% RSLogix 500 project Intro to PLC Job HO4 Greg.RSS, saved by version 10.00.00.00 %
PROJECT "UNTITLED"    % processor: Bul.1763 MicroLogix 1100 Series B %

PROGRAM FILES
  LAD 2   9 rungs

DATA FILES
  O0 OUTPUT  4 elements
  I1 INPUT  6 elements
  S2 STATUS  66 elements
  B3 BINARY  1 elements
  T4 TIMER  1 elements
  C5 COUNTER  1 elements
  R6 CONTROL  1 elements
  N7 INTEGER  1 elements
  F8 FLOAT  1 elements

LADDER 2
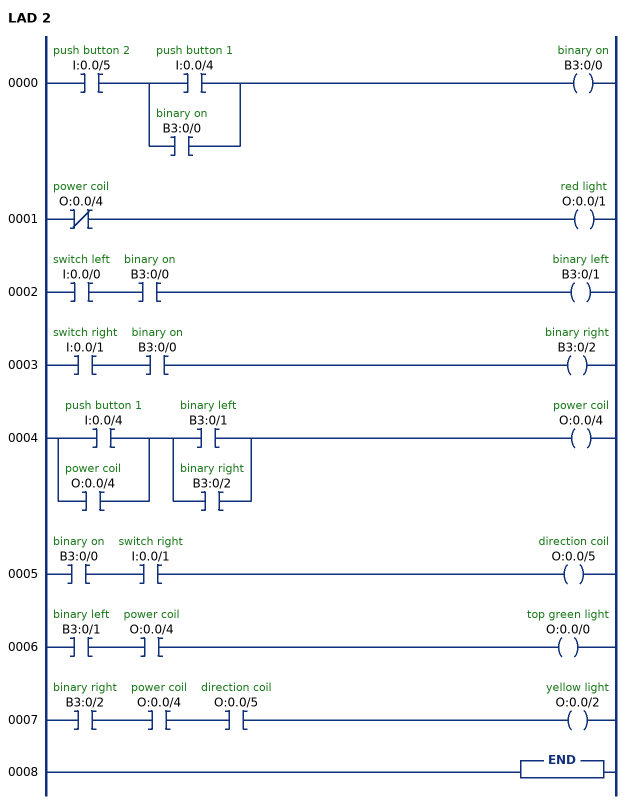
% Rung: 0 %
SOR XIC I:0.0/5 BST XIC I:0.0/4 NXB XIC B3:0/0 BND OTE B3:0/0 EOR
%   I:0.0/5  "push button 2" %
%   I:0.0/4  "push button 1" %
%   B3:0/0  "binary on" %
% Rung: 1 %
SOR XIO O:0.0/4 OTE O:0.0/1 EOR
%   O:0.0/4  "power coil" %
%   O:0.0/1  "red light" %
% Rung: 2 %
SOR XIC I:0.0/0 XIC B3:0/0 OTE B3:0/1 EOR
%   I:0.0/0  "switch left" %
%   B3:0/0  "binary on" %
%   B3:0/1  "binary left" %
% Rung: 3 %
SOR XIC I:0.0/1 XIC B3:0/0 OTE B3:0/2 EOR
%   I:0.0/1  "switch right" %
%   B3:0/0  "binary on" %
%   B3:0/2  "binary right" %
% Rung: 4 %
SOR BST XIC I:0.0/4 NXB XIC O:0.0/4 BND BST XIC B3:0/1 NXB XIC B3:0/2 BND OTE O:0.0/4 EOR
%   I:0.0/4  "push button 1" %
%   O:0.0/4  "power coil" %
%   B3:0/1  "binary left" %
%   B3:0/2  "binary right" %
% Rung: 5 %
SOR XIC B3:0/0 XIC I:0.0/1 OTE O:0.0/5 EOR
%   B3:0/0  "binary on" %
%   I:0.0/1  "switch right" %
%   O:0.0/5  "direction coil" %
% Rung: 6 %
SOR XIC B3:0/1 XIC O:0.0/4 OTE O:0.0/0 EOR
%   B3:0/1  "binary left" %
%   O:0.0/4  "power coil" %
%   O:0.0/0  "top green light" %
% Rung: 7 %
SOR XIC B3:0/2 XIC O:0.0/4 XIC O:0.0/5 OTE O:0.0/2 EOR
%   B3:0/2  "binary right" %
%   O:0.0/4  "power coil" %
%   O:0.0/5  "direction coil" %
%   O:0.0/2  "yellow light" %
% Rung: 8 %
SOR END EOR

OTHER DOCUMENTED ADDRESSES
  B3:0/5  "direction coil"
  C5:0  "counter"
  C5:0.ACC  "move"
  C5:0.ACC/0  "counter acc"
  C5:0/DN  "counter done"
  N7:0  "integer"
